FUNCTION_BLOCK FB_LightDancer
VAR_INPUT
	Execute:BOOL;
	Terminate:BOOL;
END_VAR
VAR_OUTPUT
	Done,
	Busy,
	Error:BOOL;
	Light:ARRAY[1..9]	OF	BOOL;
END_VAR
VAR
	STATE: FunctionBlockStates;//at startup initialises to 0;
	counter: INT;
	i: INT;
	cyclecounter: INT;
END_VAR

CASE	STATE	OF
	FunctionBlockStates.Idle://Idle
		Done:=
		Busy:=
		Error:=FALSE;
		counter:=
		cyclecounter:=0;
		IF	Execute	THEN
			STATE:=FunctionBlockStates.Busy;
			busy:=TRUE;
		END_IF
	FunctionBlockStates.Busy://Busy
	
		IF	counter>9	THEN
			counter:=0;
			cyclecounter:=cyclecounter+1;
		END_IF
		IF	NOT Terminate	THEN
			IF	cyclecounter<>5 	THEN
				CASE	counter	OF
					0:
						FOR	i:=1	TO	9	DO
							Light[i]:=FALSE;
						END_FOR
					ELSE
						Light[counter]:=TRUE;
						
//						FOR	i:=1	TO	9	DO
//							IF	i<>counter	THEN
//								Light[i]:=FALSE;
//							END_IF
//						END_FOR
				END_CASE
				counter:=counter+1;
			ELSE
				state:=FunctionBlockStates.Done;
		END_IF
		ELSE
			state:=FunctionBlockStates.Error;
		END_IF
	FunctionBlockStates.Done://Done
		Done:=TRUE;
		Busy:=FALSE;
		IF	Execute=FALSE	THEN
			state:=FunctionBlockStates.Idle;
		END_IF
	FunctionBlockStates.Error://Error
		Error:=TRUE;
		Busy:=FALSE;
		IF	Execute=FALSE	THEN
			state:=FunctionBlockStates.Idle;
		END_IF
END_CASE

END_FUNCTION_BLOCK

(* stored: Version 1.1.0.1, ProductVersion 3.1.4024.11
   POU FB_LightDancer: Id {ddaef838-42fd-4d52-9361-898250b9fff8}, SpecialFunc None *)
